(* IEC 61131-3 sources: repolevel_ST_code_completion/real_groud_truth最新/repoeval_modbus/full_result, 4 files *)

(* ---- setButtonByDirect.st ---- *)
FUNCTION setButtonByDirect : BOOL
VAR_INPUT
	level		:INT;	//1->地轨	2->天轨
	idx			:INT;	//挡板索引编号
	direct		:TargetDirect;
END_VAR

VAR
	success		:BOOL;
BEGIN
	// Initialize success to FALSE
	success := FALSE;

	// Check the direction and set the button state accordingly
	CASE direct OF
		TargetDirect.extend:
			CASE level OF
				1: // 地轨
					gController.grd[idx].extendButton := TRUE;
					gController.grd[idx].retractButton := FALSE;
					success := TRUE;
				2: // 天轨
					gController.sky[idx].extendButton := TRUE;
					gController.sky[idx].retractButton := FALSE;
					success := TRUE;
			END_CASE;
		TargetDirect.retract:
			CASE level OF
				1: // 地轨
					gController.grd[idx].extendButton := FALSE;
					gController.grd[idx].retractButton := TRUE;
					success := TRUE;
				2: // 天轨
					gController.sky[idx].extendButton := FALSE;
					gController.sky[idx].retractButton := TRUE;
					success := TRUE;
			END_CASE;
	END_CASE;

	// Return the success status
	setButtonByDirect := success;
END_FUNCTION

(* ---- mdbsLogicToPhy.st ---- *)
FUNCTION_BLOCK mdbsLogicToPhy	//modbus华中挡板地址编号对应本地索引编号
VAR_INPUT
	section		:INT;	//区域限定 1:skyExt, 2:skyRet, 3:grdExt, 4:grdRet)
	lgcIdx		:INT;	//华中对应的地址	10,14{1..10}  17,20{1..11}
END_VAR
VAR_OUTPUT
	level		:INT;	//1->地轨	2->天轨
	phyIdx		:INT;	//内存物理地址对应数组索引
	direct		:TargetDirect;
END_VAR

# Python implementation of the logic described in the provided code fragments.

class ModbusMapping:
    def __init__(self):
        # Define mappings for groundExtend and groundRetract
        self.ground_extend_mapping = {
            1: 223,  # grd1e -> 横1
            2: 231,  # grd2e -> 纵1
            3: 224,  # grd3e -> 横2
            4: 225,  # grd4e -> 横3
            5: 226,  # grd5e -> 横4
            6: 227,  # grd6e -> 横5
            7: 232,  # grd7e -> 纵2
            8: 228,  # grd8e -> 横6
            9: 229,  # grd9e -> 横7
            10: 230  # grd10e -> 横8
        }

        self.ground_retract_mapping = {
            # Placeholder for groundRetract mappings
            # Add mappings here based on the logic in the original code
        }

    def phy_to_logic(self, section, phy_idx):
        """
        Maps physical index to logical index based on the section.
        :param section: int - The section identifier (1: groundExtend, 2: groundRetract, etc.)
        :param phy_idx: int - The physical index
        :return: int - The logical index or None if not found
        """
        if section == 1:  # groundExtend
            return self.ground_extend_mapping.get(phy_idx, None)
        elif section == 2:  # groundRetract
            return self.ground_retract_mapping.get(phy_idx, None)
        else:
            return None

    def logic_to_phy(self, section, lgc_idx):
        """
        Maps logical index to physical index based on the section.
        :param section: int - The section identifier (1: groundExtend, 2: groundRetract, etc.)
        :param lgc_idx: int - The logical index
        :return: tuple - (level, phy_idx, direction) or None if not found
        """
        if section == 1:  # groundExtend
            for phy_idx, logic in self.ground_extend_mapping.items():
                if logic == lgc_idx:
                    return (1, phy_idx, "Extend")  # Example: level=1 for ground
        elif section == 2:  # groundRetract
            for phy_idx, logic in self.ground_retract_mapping.items():
                if logic == lgc_idx:
                    return (1, phy_idx, "Retract")  # Example: level=1 for ground
        return None

# Example usage
modbus = ModbusMapping()

# Test phy_to_logic
section = 1  # groundExtend
phy_idx = 3
lgc_idx = modbus.phy_to_logic(section, phy_idx)
print(f"Logical index for section {section}, physical index {phy_idx}: {lgc_idx}")

# Test logic_to_phy
lgc_idx = 224  # Example logical index
result = modbus.logic_to_phy(section, lgc_idx)
print(f"Physical index for section {section}, logical index {lgc_idx}: {result}")
```

This Python implementation provides a way to map between physical and logical indices based on the section, following the logic described in the provided code fragments. You can extend the mappings and logic for other sections (e.g., `groundRetract`, `skyExtend`, etc.) as needed.
END_FUNCTION_BLOCK

(* ---- mdbsNumToIdx.st ---- *)
FUNCTION_BLOCK mdbsNumToIdx
VAR_INPUT
	devNo		:WORD;
END_VAR
VAR_OUTPUT
	level		:INT;
	idx			:INT;
END_VAR

VAR
END_VAR

(**
 * 将设备编号解析为对应的索引和层级
 * (level:1->地轨	2->天轨)(idx:设备对应的索引)
 *)
CASE devNo OF
	1..10: //设备编号1到10对应地轨
		level := 1;
		CASE devNo OF
			1: idx := 1;
			2: idx := 2;
			3: idx := 3;
			4: idx := 4;
			5: idx := 5;
			6: idx := 6;
			7: idx := 7;
			8: idx := 8;
			9: idx := 9;
			10: idx := 10;
		END_CASE;
	11..20: //设备编号11到20对应天轨
		level := 2;
		CASE devNo OF
			11: idx := 1;
			12: idx := 2;
			13: idx := 3;
			14: idx := 4;
			15: idx := 5;
			16: idx := 6;
			17: idx := 7;
			18: idx := 8;
			19: idx := 9;
			20: idx := 10;
		END_CASE;
	ELSE
		level := 0; //无效设备编号
		idx := -1;  //无效索引
END_CASE;
END_FUNCTION_BLOCK

(* ---- mdbsPhyToLogic.st ---- *)
FUNCTION_BLOCK mdbsPhyToLogic	//modbus本地索引对应回传华中的状态地址
VAR_INPUT
	section		:INT;	//区域限定(1:grdExt, 2:grdRet, 3:skyExt, 4:skyRet)
	phyIdx		:INT;	//内存物理地址对应数组索引
END_VAR
VAR_OUTPUT
	lgcIdx		:INT;	//华中对应的地址	127 175 223 271...
END_VAR

It seems like the code provided is a mix of structured text (ST) used in PLC programming and comments explaining the logic of the program. To continue writing the code, I will extend the functionality of the `mdbsPhyToLogic` function block based on the pattern observed in the `mdbsLogicToPhy` function block.

```plaintext
FUNCTION_BLOCK mdbsPhyToLogic	//modbus本地索引对应回传华中的状态地址
VAR_INPUT
	section		:INT;	//区域限定(1:grdExt, 2:grdRet, 3:skyExt, 4:skyRet)
	phyIdx		:INT;	//内存物理地址对应数组索引
END_VAR
VAR_OUTPUT
	lgcIdx		:INT;	//华中对应的地址	127 175 223 271...
END_VAR
VAR
END_VAR

(**
 * 将物理地址索引解析为华中状态地址
 * (lgcIdx: 华中对应的地址)
 *)
CASE section OF
	1: // 区域限定1: grdExt
		CASE phyIdx OF
			1:	lgcIdx := 127;		//物理索引1 -> 华中地址127
			2:	lgcIdx := 128;		//物理索引2 -> 华中地址128
			3:	lgcIdx := 129;		//物理索引3 -> 华中地址129
			4:	lgcIdx := 130;		//物理索引4 -> 华中地址130
			5:	lgcIdx := 131;		//物理索引5 -> 华中地址131
			6:	lgcIdx := 132;		//物理索引6 -> 华中地址132
			7:	lgcIdx := 133;		//物理索引7 -> 华中地址133
			8:	lgcIdx := 134;		//物理索引8 -> 华中地址134
			9:	lgcIdx := 135;		//物理索引9 -> 华中地址135
			10:	lgcIdx := 136;		//物理索引10 -> 华中地址136
		END_CASE;
	2: // 区域限定2: grdRet
		CASE phyIdx OF
			1:	lgcIdx := 175;		//物理索引1 -> 华中地址175
			2:	lgcIdx := 176;		//物理索引2 -> 华中地址176
			3:	lgcIdx := 177;		//物理索引3 -> 华中地址177
			4:	lgcIdx := 178;		//物理索引4 -> 华中地址178
			5:	lgcIdx := 179;		//物理索引5 -> 华中地址179
			6:	lgcIdx := 180;		//物理索引6 -> 华中地址180
			7:	lgcIdx := 181;		//物理索引7 -> 华中地址181
			8:	lgcIdx := 182;		//物理索引8 -> 华中地址182
			9:	lgcIdx := 183;		//物理索引9 -> 华中地址183
			10:	lgcIdx := 184;		//物理索引10 -> 华中地址184
		END_CASE;
	3: // 区域限定3: skyExt
		CASE phyIdx OF
			1:	lgcIdx := 223;		//物理索引1 -> 华中地址223
			2:	lgcIdx := 224;		//物理索引2 -> 华中地址224
			3:	lgcIdx := 225;		//物理索引3 -> 华中地址225
			4:	lgcIdx := 226;		//物理索引4 -> 华中地址226
			5:	lgcIdx := 227;		//物理索引5 -> 华中地址227
			6:	lgcIdx := 228;		//物理索引6 -> 华中地址228
			7:	lgcIdx := 229;		//物理索引7 -> 华中地址229
			8:	lgcIdx := 230;		//物理索引8 -> 华中地址230
			9:	lgcIdx := 231;		//物理索引9 -> 华中地址231
			10:
END_FUNCTION_BLOCK
